FUNCTION_BLOCK MECH_VIEW (* View of a Linear Mechanism *)
  (* Standard: 61499-1; Classification: View *)
  (* Version 0.0, 2002-04-05, JHC, Rockwell Automation, Copied/Modified from CNV_VIEW *)
  (* Compiler header: package fb.rt.hmi; *)
  (* Compiler classdef: public class MECH_VIEW extends XABS_VIEW *)
  (* Compiler Java IBM VisualAge 3.0 *)
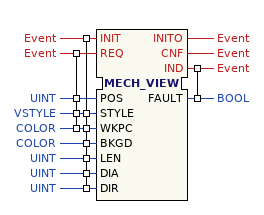
  EVENT_INPUT
    INIT WITH STYLE, WKPC, BKGD, LEN, DIA, DIR; (* Initialize *)
    REQ WITH POS, STYLE, WKPC; (* Update the display *)
  END_EVENT
  EVENT_OUTPUT
    INITO; (* Initialized *)
    CNF; (* Display Updated *)
    IND WITH FAULT; (* Change in FAULT status *)
  END_EVENT
  VAR_INPUT
    POS : UINT; (* Mechanism displacement *)
    STYLE : VSTYLE := RING; (* View style *)
    WKPC : COLOR := blue; (* Foreground Color *)
    BKGD : COLOR := blue; (* Background Color *)
    LEN : UINT; (* Length in Diameters *)
    DIA : UINT; (* Diameter *)
    DIR : UINT; (* Orientation:0=L/R,1=T/B,2=R/L,3=B/T *)
  END_VAR
  VAR_OUTPUT
    FAULT : BOOL; (* 0=Normal,1=Fault *)
  END_VAR
END_FUNCTION_BLOCK
